// TIA Portal V20 export
DATA_BLOCK "GDB_Control"   // DB
TITLE = GDB_Control (minimal)
{ S7_Optimized_Access := 'TRUE' }
// Minimal control DB for ABCDE 5-point cycle. Holds kinematic enable/home arrays + mirror status. Trimmed from v9 (palletizing/recipe/manual fields removed).
   VAR
      enableAxes : Bool;   // Enable kinematic group via LKinCtrl_MC_GroupPower
      axesEnabled : Bool;   // Status: all axes enabled (mirror from MC_GroupPower.axesEnabled)
      resetAxes : Bool;   // Reset kinematic group via LKinCtrl_MC_GroupReset
   END_VAR
   VAR RETAIN
      axesError : Bool;   // Status: error on any joint TO
   END_VAR
   VAR
      homeAxes : Bool;   // Home kinematic group via LKinCtrl_MC_GroupHome
      axesHomed : Bool;   // Status: all 4 joint TOs report StatusWord.X5 (Homed)
      robotStandstill : Bool;   // Status: all 4 joint TOs report StatusWord.X7 (Standstill)
   END_VAR
   VAR RETAIN
      HomePos : Array[1..6] of LReal;   // Home positions per kinematic axis index (A1=J1, A2=J3, A3=J2, A4=J4). Initialized by Startup.scl.
   END_VAR
   VAR
      HomeMode : Array[1..6] of Int;   // Home mode per kinematic axis index. 7 = set actual position (no physical homing motion).
      StartMode : Array[1..6] of DInt;   // Start mode for MC_Power per axis. 1 = enable position-controlled. Initialized by Startup.scl to avoid retain-drift issues.
      StopMode : Array[1..6] of Int;   // Stop mode for MC_Power per axis. 1 = immediate stop. Initialized by Startup.scl.
      RestartMode : Array[1..7] of Bool;   // Restart mode flags for MC_GroupReset per axis.
   END_VAR
BEGIN
END_DATA_BLOCK
